Fanuc KAREL source: NC0007.KL

-- PROVISIONAL review KL for V940-1; original PC SHA256 f89210e89de55c96493db2aa72f8ba0977cfdfd8a699ca81ac3331224fbe6bae
-- Incomplete behavior may be omitted. Consult companion uncertainty JSON. Do not deploy.
PROGRAM NC0007
%NOLOCKGROUP
-- UNRESOLVED_LOCAL_POOL 1 cells at code offset 3; source declarations unknown
-- DIRECT_LOCAL_WORD_ACCESS alone does not prove INTEGER, REAL, or BOOLEAN
BEGIN
  -- V9_EXPOSED_INDEXED_TABLE_HINT layout=0001; 20 counted words exposed once; source arms/runtime held
  -- V9_CONDITION_STACK_HINT 10 bounded expression windows; static native code-base-relative target link; source arms held
  -- UNRESOLVED_PC offsets 0-8; opcodes 2B,2C,7B
  -- UNRESOLVED_PC offsets 13-20; opcodes 9D,23
  -- UNRESOLVED_PC offsets 25-38; opcodes 21,9D,57,79
  -- UNRESOLVED_PC offsets 43-56; opcodes 21,9D,57,79
  -- UNRESOLVED_PC offsets 61-74; opcodes 21,9D,57,79
  -- UNRESOLVED_PC offsets 79-92; opcodes 21,9D,57,79
  -- UNRESOLVED_PC offsets 97-110; opcodes 21,9D,57,79
  -- UNRESOLVED_PC offsets 115-128; opcodes 21,9D,57,79
  -- UNRESOLVED_PC offsets 133-146; opcodes 21,9D,57,79
  -- UNRESOLVED_PC offsets 151-164; opcodes 21,9D,57,79
  -- UNRESOLVED_PC offsets 169-182; opcodes 21,9D,57,79
  -- UNRESOLVED_PC offsets 187-200; opcodes 21,9D,57,79
  -- UNRESOLVED_PC offsets 205-219; opcodes 21,9D,52,23
  -- UNRESOLVED_PC offsets 224-229; opcodes 7A
  -- UNRESOLVED_PC offsets 234-252; opcodes 21,2E,52,23
  -- UNRESOLVED_PC offsets 262-267; opcodes 7A
  -- UNRESOLVED_PC offsets 272-290; opcodes 21,2E,52,23
  -- UNRESOLVED_PC offsets 300-305; opcodes 7A
  -- UNRESOLVED_PC offsets 310-328; opcodes 21,2E,52,23
  -- UNRESOLVED_PC offsets 338-343; opcodes 7A
  -- UNRESOLVED_PC offsets 348-366; opcodes 21,2E,52,23
  -- UNRESOLVED_PC offsets 376-381; opcodes 7A
  -- UNRESOLVED_PC offsets 386-404; opcodes 21,2E,52,23
  -- UNRESOLVED_PC offsets 414-419; opcodes 7A
  -- UNRESOLVED_PC offsets 424-442; opcodes 21,2E,52,23
  -- UNRESOLVED_PC offsets 452-457; opcodes 7A
  -- UNRESOLVED_PC offsets 462-480; opcodes 21,2E,52,23
  -- UNRESOLVED_PC offsets 490-495; opcodes 7A
  -- UNRESOLVED_PC offsets 500-518; opcodes 21,2E,52,23
  -- UNRESOLVED_PC offsets 528-533; opcodes 7A
  -- UNRESOLVED_PC offsets 538-556; opcodes 21,2E,52,23
  -- UNRESOLVED_PC offsets 566-571; opcodes 7A
  -- UNRESOLVED_PC offsets 576-594; opcodes 21,2E,52,23
  -- UNRESOLVED_PC offsets 604-608; opcodes 7F
  -- UNRESOLVED_PC offsets 613-617; opcodes 27,AA
  -- UNRESOLVED_PC offsets 622-626; opcodes 7F
END NC0007
